PROGRAM Godot
VAR
	on : BOOL;
	//_Godot : GodotHmi(Main.Movers[1]);
END_VAR

IF NOT on THEN
	RETURN;
END_IF

//_Godot.CyclicLogic();

END_PROGRAM

(* stored: Version 1.1.0.1, ProductVersion 3.1.4026.19
   POU Godot: Id {25ca116f-cc26-4fba-af85-d3cc1123b179}, SpecialFunc None *)
